// TIA Portal V19 export
DATA_BLOCK "MES_Send_Buffer_Msg_Topic4XX"   // DB30
// stored: Access Published, MemoryReserve 100
   VAR RETAIN
      lastId : DInt;   // id ultimo messaggio inviato
      "Counter" : DInt;   // contatore messaggi da inviare
      msg : Array[1.."MES_MSG_ITEMS"] of "MES_Msg";   // buffer dei messaggi da inviare
   END_VAR
BEGIN
END_DATA_BLOCK
